{attribute 'GeneratedUsingTerminal: EK1100-0000-0018'}
{attribute addProperty BoxType "EK1100-0000-0018"}
{attribute addProperty Id "Beckhoff_EP6xxxEK1122Beckhoff_EP6xxxEK1122_1419FDD91410"}
{attribute addProperty CRC "3775435886"}
{attribute addProperty Size "1410"}
TYPE Beckhoff_EP6xxx_E108946E EXTENDS EK1100_AB5A9467 :
STRUCT
	{attribute addProperty Name "Beckhoff_EP6xxxEK1122"}
	Beckhoff_EP6xxxEK1122 : Beckhoff_EP6xxxEK1122_1419FDD9;
END_STRUCT
END_TYPE

(* stored: Version 1.2.0.0, ProductVersion 3.1.4024.9
   DUT Beckhoff_EP6xxx_E108946E: Id {f6ab4780-af50-4b42-ba9d-957960776349} *)
